(* IEC 61131-3 sources: plc_on_fpga_riscv_hybrid/RV_FPGA_PLC_IDE_Projects/Arithmatic_MUL, 1 file *)

(* ---- Arithmatic_MUL.il ---- *)
VAR
    Add_Res   : INT
END_VAR

PROGRAM Arithmatic_MUL
    Addition :
        LD     %SW.0
        MUL    %SW.1
        MUL    %SW.2
        MUL    %SW.3
        MUL    %SW.4
        ST     %LEDG.0
END_PROGRAM
